// TIA Portal V18 export
// export: Created 2026-03-12T16:04:35.9081085Z, ExportSetting WithDefaults, DisplayName Totally Integrated Automation Portal, DisplayVersion V18 Update 5, DisplayName TIA Portal Openness, DisplayVersion V18 Update 5, DisplayName TIA Portal Version Control Interface, DisplayVersion V18, DisplayName SINAMICS Startdrive Advanced, DisplayVersion V18, DisplayName SINAMICS Startdrive G130, G150, S120, S150, SINAMICS MV, S210, DisplayVersion V18, DisplayName SINAMICS Startdrive G110M, G120, G120C, G120D, G120P, G115D, DisplayVersion V18, DisplayName STEP 7 Professional, DisplayVersion V18 Update 5, DisplayName STEP 7 Safety, DisplayVersion V18, DisplayName WinCC Professional, DisplayVersion V18 Update 5
FUNCTION_BLOCK "FB_MOVE_SKID_DESAGUAMENTO"   // FB37, LAD
{ S7_Optimized_Access := 'TRUE' }
VERSION : 0.1
// stored: AutoNumber true, IsIECCheckEnabled false, IsRetainMemResEnabled false, MemoryReserve 100, SetENOAutomatically false, UDAEnableTagReadback false
   VAR_INPUT
      STATUS_GERAL_DWORD : Struct   // 17359 - 17383 = 26 Words
         STS_PRINCIPAL_CENTRIFUGA : DWord;   // Status do motor principal da centrífuga.0 = Desligado1 = Ligado2 = Falha
         STS_SECUNDARIO_CENTRIFUGA : DWord;   // Status do motor secundário da centrífuga.0 = Desligado1 = Ligado2 = Falha
         STS_BBA_LODO : DWord;   // Status do motor da bomba de lodo0 = Desligado1 = Ligado2 = Falha
         STS_BBA_POLIMERO : DWord;   // Status do motor da bomba de polímero0 = Desligado1 = Ligado2 = Falha
         STS_ROSCA_POLIMERO : DWord;   // Status do motor da rosca de polímero0 = Desligado1 = Ligado2 = Falha
         STS_ROSCA_LODO : DWord;   // Status do motor da rosca de lodo0 = Desligado1 = Ligado2 = Falha
         STS_AGITADOR_01 : DWord;   // Status do motor do agitador 01 do preparador de polímero0 = Desligado1 = Ligado2 = Falha
         STS_BBA_CLARIFICADOR_01 : DWord;   // Status do motor da bomba de clarificado 010 = Desligado1 = Ligado2 = Falha
         STS_BBA_CLARIFICADOR_02 : DWord;   // Status do motor da bomba de clarificado 020 = Desligado1 = Ligado2 = Falha
         STS_BBA_LAVAGEM : DWord;   // Status do motor da bomba de lavagem0 = Desligado1 = Ligado2 = Falha
         STS_AGITADOR_02 : DWord;   // Status do motor do agitador 02 do preparador de polímero0 = Desligado1 = Ligado2 = Falha
         STS_RESISTENCIA_AQUECIMENTO_POLIMERO : DWord;   // Status do motor da resistência de aquecimento de polímero0 = Desligado1 = Ligado2 = Falha
         STS_VALVULA_AGUA_ADENSADOR : DWord;   // Status da válvula de entrada de água do preparador de polímero0 = Desligado1 = Ligado
      END_STRUCT;
      INDICE : Int := 16;
   END_VAR
   VAR_OUTPUT
      STATUS_GERAL : Struct   // 17359 - 17383 = 26 Words
         STS_PRINCIPAL_CENTRIFUGA : Word;   // Status do motor principal da centrífuga.0 = Desligado1 = Ligado2 = Falha
         STS_SECUNDARIO_CENTRIFUGA : Word;   // Status do motor secundário da centrífuga.0 = Desligado1 = Ligado2 = Falha
         STS_BBA_LODO : Word;   // Status do motor da bomba de lodo0 = Desligado1 = Ligado2 = Falha
         STS_BBA_POLIMERO : Word;   // Status do motor da bomba de polímero0 = Desligado1 = Ligado2 = Falha
         STS_ROSCA_POLIMERO : Word;   // Status do motor da rosca de polímero0 = Desligado1 = Ligado2 = Falha
         STS_ROSCA_LODO : Word;   // Status do motor da rosca de lodo0 = Desligado1 = Ligado2 = Falha
         STS_AGITADOR_01 : Word;   // Status do motor do agitador 01 do preparador de polímero0 = Desligado1 = Ligado2 = Falha
         STS_BBA_CLARIFICADOR_01 : Word;   // Status do motor da bomba de clarificado 010 = Desligado1 = Ligado2 = Falha
         STS_BBA_CLARIFICADOR_02 : Word;   // Status do motor da bomba de clarificado 020 = Desligado1 = Ligado2 = Falha
         STS_BBA_LAVAGEM : Word;   // Status do motor da bomba de lavagem0 = Desligado1 = Ligado2 = Falha
         STS_AGITADOR_02 : Word;   // Status do motor do agitador 02 do preparador de polímero0 = Desligado1 = Ligado2 = Falha
         STS_RESISTENCIA_AQUECIMENTO_POLIMERO : Word;   // Status do motor da resistência de aquecimento de polímero0 = Desligado1 = Ligado2 = Falha
         STS_VALVULA_AGUA_ADENSADOR : Word;   // Status da válvula de entrada de água do preparador de polímero0 = Desligado1 = Ligado
      END_STRUCT;
   END_VAR
BEGIN

REGION Network 1
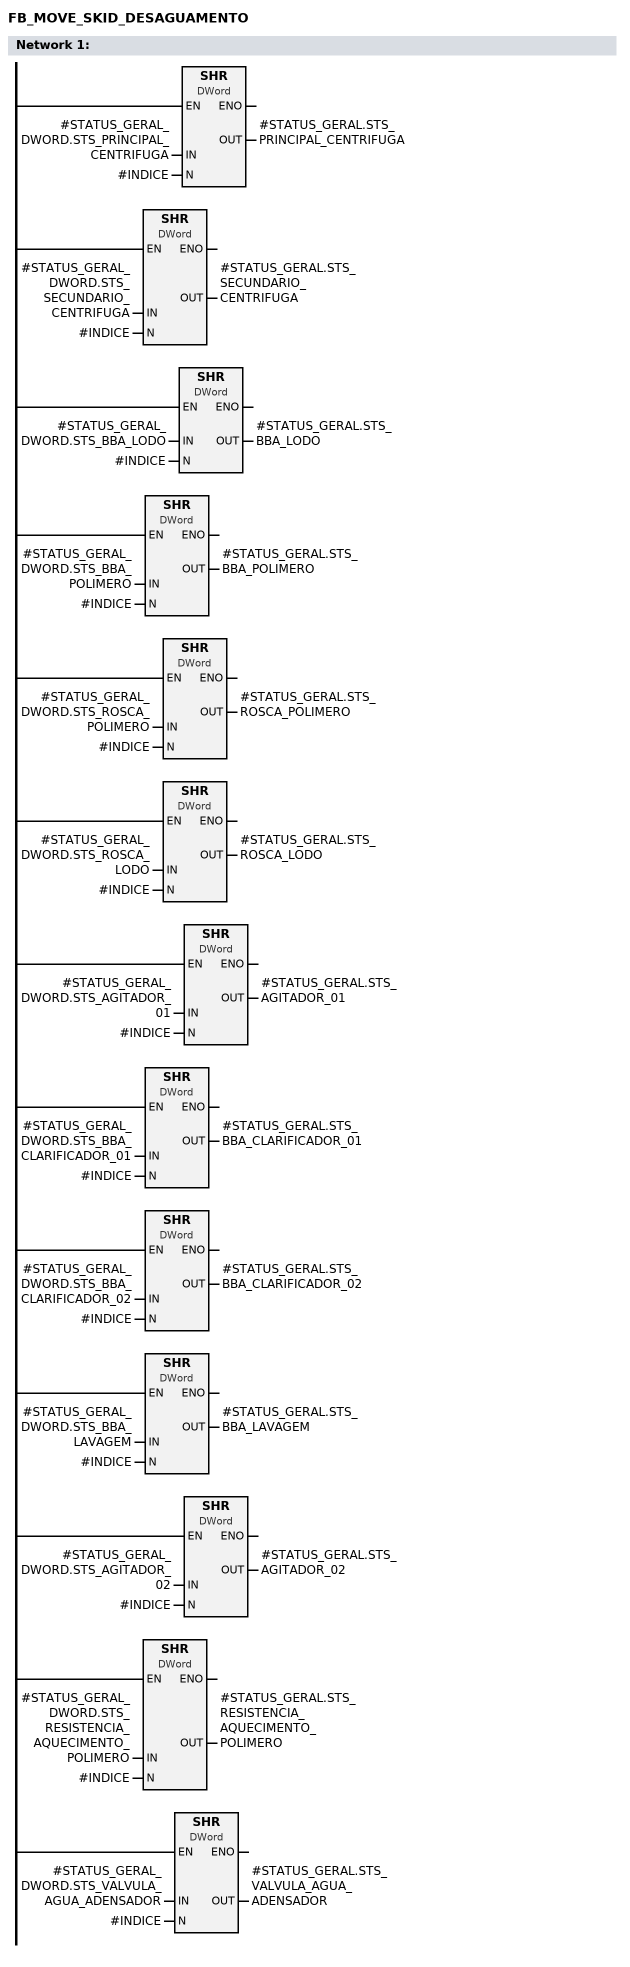
   RUNG wire#powerrail
      { S7_Templates := "SrcType := DWord" } Shr(in := #STATUS_GERAL_DWORD.STS_PRINCIPAL_CENTRIFUGA, n := #INDICE, out => #STATUS_GERAL.STS_PRINCIPAL_CENTRIFUGA)
   END_RUNG
   RUNG wire#powerrail
      { S7_Templates := "SrcType := DWord" } Shr(in := #STATUS_GERAL_DWORD.STS_SECUNDARIO_CENTRIFUGA, n := #INDICE, out => #STATUS_GERAL.STS_SECUNDARIO_CENTRIFUGA)
   END_RUNG
   RUNG wire#powerrail
      { S7_Templates := "SrcType := DWord" } Shr(in := #STATUS_GERAL_DWORD.STS_BBA_LODO, n := #INDICE, out => #STATUS_GERAL.STS_BBA_LODO)
   END_RUNG
   RUNG wire#powerrail
      { S7_Templates := "SrcType := DWord" } Shr(in := #STATUS_GERAL_DWORD.STS_BBA_POLIMERO, n := #INDICE, out => #STATUS_GERAL.STS_BBA_POLIMERO)
   END_RUNG
   RUNG wire#powerrail
      { S7_Templates := "SrcType := DWord" } Shr(in := #STATUS_GERAL_DWORD.STS_ROSCA_POLIMERO, n := #INDICE, out => #STATUS_GERAL.STS_ROSCA_POLIMERO)
   END_RUNG
   RUNG wire#powerrail
      { S7_Templates := "SrcType := DWord" } Shr(in := #STATUS_GERAL_DWORD.STS_ROSCA_LODO, n := #INDICE, out => #STATUS_GERAL.STS_ROSCA_LODO)
   END_RUNG
   RUNG wire#powerrail
      { S7_Templates := "SrcType := DWord" } Shr(in := #STATUS_GERAL_DWORD.STS_AGITADOR_01, n := #INDICE, out => #STATUS_GERAL.STS_AGITADOR_01)
   END_RUNG
   RUNG wire#powerrail
      { S7_Templates := "SrcType := DWord" } Shr(in := #STATUS_GERAL_DWORD.STS_BBA_CLARIFICADOR_01, n := #INDICE, out => #STATUS_GERAL.STS_BBA_CLARIFICADOR_01)
   END_RUNG
   RUNG wire#powerrail
      { S7_Templates := "SrcType := DWord" } Shr(in := #STATUS_GERAL_DWORD.STS_BBA_CLARIFICADOR_02, n := #INDICE, out => #STATUS_GERAL.STS_BBA_CLARIFICADOR_02)
   END_RUNG
   RUNG wire#powerrail
      { S7_Templates := "SrcType := DWord" } Shr(in := #STATUS_GERAL_DWORD.STS_BBA_LAVAGEM, n := #INDICE, out => #STATUS_GERAL.STS_BBA_LAVAGEM)
   END_RUNG
   RUNG wire#powerrail
      { S7_Templates := "SrcType := DWord" } Shr(in := #STATUS_GERAL_DWORD.STS_AGITADOR_02, n := #INDICE, out => #STATUS_GERAL.STS_AGITADOR_02)
   END_RUNG
   RUNG wire#powerrail
      { S7_Templates := "SrcType := DWord" } Shr(in := #STATUS_GERAL_DWORD.STS_RESISTENCIA_AQUECIMENTO_POLIMERO, n := #INDICE, out => #STATUS_GERAL.STS_RESISTENCIA_AQUECIMENTO_POLIMERO)
   END_RUNG
   RUNG wire#powerrail
      { S7_Templates := "SrcType := DWord" } Shr(in := #STATUS_GERAL_DWORD.STS_VALVULA_AGUA_ADENSADOR, n := #INDICE, out => #STATUS_GERAL.STS_VALVULA_AGUA_ADENSADOR)
   END_RUNG
   // the same network as SCL:
   #STATUS_GERAL.STS_PRINCIPAL_CENTRIFUGA := SHR(IN := #STATUS_GERAL_DWORD.STS_PRINCIPAL_CENTRIFUGA, N := #INDICE);
   #STATUS_GERAL.STS_SECUNDARIO_CENTRIFUGA := SHR(IN := #STATUS_GERAL_DWORD.STS_SECUNDARIO_CENTRIFUGA, N := #INDICE);
   #STATUS_GERAL.STS_BBA_LODO := SHR(IN := #STATUS_GERAL_DWORD.STS_BBA_LODO, N := #INDICE);
   #STATUS_GERAL.STS_BBA_POLIMERO := SHR(IN := #STATUS_GERAL_DWORD.STS_BBA_POLIMERO, N := #INDICE);
   #STATUS_GERAL.STS_ROSCA_POLIMERO := SHR(IN := #STATUS_GERAL_DWORD.STS_ROSCA_POLIMERO, N := #INDICE);
   #STATUS_GERAL.STS_ROSCA_LODO := SHR(IN := #STATUS_GERAL_DWORD.STS_ROSCA_LODO, N := #INDICE);
   #STATUS_GERAL.STS_AGITADOR_01 := SHR(IN := #STATUS_GERAL_DWORD.STS_AGITADOR_01, N := #INDICE);
   #STATUS_GERAL.STS_BBA_CLARIFICADOR_01 := SHR(IN := #STATUS_GERAL_DWORD.STS_BBA_CLARIFICADOR_01, N := #INDICE);
   #STATUS_GERAL.STS_BBA_CLARIFICADOR_02 := SHR(IN := #STATUS_GERAL_DWORD.STS_BBA_CLARIFICADOR_02, N := #INDICE);
   #STATUS_GERAL.STS_BBA_LAVAGEM := SHR(IN := #STATUS_GERAL_DWORD.STS_BBA_LAVAGEM, N := #INDICE);
   #STATUS_GERAL.STS_AGITADOR_02 := SHR(IN := #STATUS_GERAL_DWORD.STS_AGITADOR_02, N := #INDICE);
   #STATUS_GERAL.STS_RESISTENCIA_AQUECIMENTO_POLIMERO := SHR(IN := #STATUS_GERAL_DWORD.STS_RESISTENCIA_AQUECIMENTO_POLIMERO, N := #INDICE);
   #STATUS_GERAL.STS_VALVULA_AGUA_ADENSADOR := SHR(IN := #STATUS_GERAL_DWORD.STS_VALVULA_AGUA_ADENSADOR, N := #INDICE);
END_REGION
END_FUNCTION_BLOCK
